FUNCTION_BLOCK ParameterSet IMPLEMENTS I_ParameterPosition
VAR
	{attribute 'hide'}
	_Position : LREAL;
END_VAR

PROPERTY Position : LREAL
GET
Position := _Position;
END_GET
SET
_Position := Position;
END_SET
END_PROPERTY

END_FUNCTION_BLOCK

(* stored: Version 1.1.0.1
   POU ParameterSet: Id {ff106fc1-0178-45a0-9307-0950a21d68af}, SpecialFunc None
   Property Position: Id {db9a9f4e-eede-465b-b1ab-a7ba37c55d35}
   Get Get: Id {f3051efa-505e-4b65-bbc1-d2e26f2f2425}
   Set Set: Id {87a37641-a65d-456c-b671-9daeefcb0dbd} *)
